Fanuc KAREL source: kf00051.KL

PROGRAM KF00051
%STACKSIZE=65535
%PRIORITY=65535
%NOLOCKGROUP
VAR
I : INTEGER
J : INTEGER
X : REAL
Y : REAL
B : BOOLEAN
C : BOOLEAN
TXT : STRING[80]
TXT2 : STRING[80]
AI : ARRAY[4] OF INTEGER
BI : ARRAY[4] OF INTEGER
P : XYZWPR
JP : JOINTPOS9
PF : POSITION
STATUS : INTEGER
-- UNRESOLVED DECLARATIONS (source type spelling not recovered)
-- V1 : TYPE_0x0013 (type_u16=0x0013)
-- V2 : TYPE_0x0013 (type_u16=0x0013)
BEGIN
-- UNRESOLVED_PC line 21 opcodes [2E 23 9F 9D 22 7A] marker_code=0
J=(J + I)
-- UNRESOLVED_PC line 23 opcodes [45 2C 23] marker_code=58
END KF00051
